# B&R Automation Studio project Test
Automation Studio 4.7.2.98

## Configuration Config1

### Task classes (Cpu.sw)
```

```

### Hardware
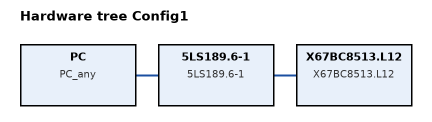
```
5LS189.6-1 : 5LS189.6-1 v1.4.0.0  [SL -> PC.SL1]
PC : PC_any v1.1.0.0 (OrderNumber=PC)
  ConfigurationID = Test_Config1
X67BC8513.L12 : X67BC8513.L12 v2.9.3.0  [PLK1 -> 5LS189.6-1.IF2 [Cable Type=PowerlinkCable, Length=10, Version=1.0.0.2]]
```

## Logical view

### Program Logical/Test (IEC)

#### Variables.var
```iecst
VAR
	TestINT : USINT;
END_VAR
```

#### Main.st
```iecst
PROGRAM _INIT
	(* Insert code here *)

END_PROGRAM

PROGRAM _CYCLIC
	TestINT := TestINT + 1;

END_PROGRAM

PROGRAM _EXIT
	(* Insert code here *)

END_PROGRAM
```

Listed in the project but not available here: Logical/Global.typ, Logical/Global.var, Logical/Libraries
